TEXTLIST GlobalPositions
  1 = 'Fold'
  2 = 'Home'
  3 = 'Approach'
  4 = 'Origin'
   = ''
END_TEXTLIST

(* stored: Version 1.1.0.1, ProductVersion 3.1.4024.10
   TextList GlobalPositions: Id {10ae2478-13c6-49bd-bb1d-4616325ba0cc} *)
